FUNCTION_BLOCK C_1Event_5States_NoConitions (* Basic FB with empty ECC *)
  (* Standard: 61499-2 *)
  (* Version 1.0, 2023-09-22, AK124910 *)
  PACKAGE servSeq;
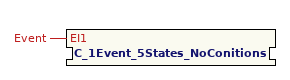
  EVENT_INPUT
    EI1;
  END_EVENT
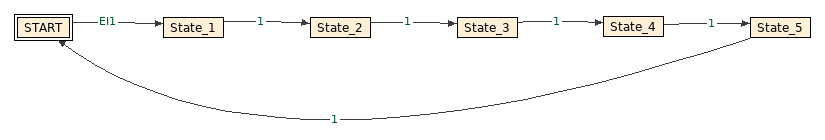
  EC_STATES
    START; (* Initial State *)
    State_1;
    State_2;
    State_3;
    State_4;
    State_5;
  END_STATES
  EC_TRANSITIONS
    START TO State_1 := EI1;
    State_1 TO State_2 := 1;
    State_2 TO State_3 := 1;
    State_3 TO State_4 := 1;
    State_4 TO State_5 := 1;
    State_5 TO START := 1;
  END_TRANSITIONS
  (* Service external/internal_interface: Basic FB with empty ECC *)
END_FUNCTION_BLOCK
